(* CoDeSys 2.3.10.0 project: Test.pro *)
(* Libraries: STANDARD.LIB 5.6.98 12:03:02 *)

(* Task configuration *)
TASK Standard (PRIORITY := 0, INTERVAL := T#10ms);
	MAIN();
END_TASK

(* Global variable list: Global_Variables *)
VAR_GLOBAL
	Zielona_1 		AT 	%Q* 	:	 BOOL:= 0;
	Zielona_2 		AT 	%Q* 	:	 BOOL:= 0;
	Zielona_3 		AT 	%Q* 	:	 BOOL:= 0;
	Zielona_4 		AT 	%Q* 	:	 BOOL:= 0;

	Czerwona_1 		AT 	%Q*		:	 BOOL:= 0;
	Czerwona_2 		AT 	%Q*		:	 BOOL:= 0;
	Czerwona_3 		AT	%Q*		:	 BOOL:= 0;
	Czerwona_4 		AT 	%Q*		:	 BOOL:= 0;

	Przycisk_1 		AT 	%I*		:	BOOL;
	Przycisk_2 		AT 	%I*		: 	BOOL;
	Przycisk_3 		AT 	%I*		: 	BOOL;
	Przycisk_4 		AT 	%I*		: 	BOOL;

	RegulatorIn_1 	AT 	%I*		:	INT;
	RegulatorIn_2 	AT 	%I*		:	INT;

	RegulatorOut_1 	AT 	%Q*		:	UDINT;
	RegulatorOut_2 	AT 	%Q*		:	UDINT;

	Scale_1			AT	%Q*		:	INT;
	Scale_2			AT	%Q*		:	INT;

	Enable_1		AT	%Q*		:	BOOL;
	Enable_2		AT 	%Q*		:	BOOL;

(*	Velo_1			AT	%I*		:	LREAL;*)
(*	Velo_2			AT	%I*		:	LREAL;*)
END_VAR

(* Global variable list: TwinCAT_Configuration *)
(* Generated automatically by TwinCAT - (read only) *)
VAR_CONFIG
	.Zielona_1 AT %QX0.0 : BOOL;	(*  ~ {LinkedWith:TIID^Device 2 (EtherCAT (v2.10 only))^Term 1 (EK1100)^Zielone (EL2004)^Channel 1^Output} *)
	.Zielona_2 AT %QX0.1 : BOOL;	(*  ~ {LinkedWith:TIID^Device 2 (EtherCAT (v2.10 only))^Term 1 (EK1100)^Zielone (EL2004)^Channel 2^Output} *)
	.Zielona_3 AT %QX0.2 : BOOL;	(*  ~ {LinkedWith:TIID^Device 2 (EtherCAT (v2.10 only))^Term 1 (EK1100)^Zielone (EL2004)^Channel 3^Output} *)
	.Zielona_4 AT %QX0.3 : BOOL;	(*  ~ {LinkedWith:TIID^Device 2 (EtherCAT (v2.10 only))^Term 1 (EK1100)^Zielone (EL2004)^Channel 4^Output} *)
	.Czerwona_1 AT %QX0.4 : BOOL;	(*  ~ {LinkedWith:TIID^Device 2 (EtherCAT (v2.10 only))^Term 1 (EK1100)^Czerwone (EL2004)^Channel 1^Output} *)
	.Czerwona_2 AT %QX0.5 : BOOL;	(*  ~ {LinkedWith:TIID^Device 2 (EtherCAT (v2.10 only))^Term 1 (EK1100)^Czerwone (EL2004)^Channel 2^Output} *)
	.Czerwona_3 AT %QX0.6 : BOOL;	(*  ~ {LinkedWith:TIID^Device 2 (EtherCAT (v2.10 only))^Term 1 (EK1100)^Czerwone (EL2004)^Channel 3^Output} *)
	.Czerwona_4 AT %QX0.7 : BOOL;	(*  ~ {LinkedWith:TIID^Device 2 (EtherCAT (v2.10 only))^Term 1 (EK1100)^Czerwone (EL2004)^Channel 4^Output} *)
	.Przycisk_1 AT %IX0.0 : BOOL;	(*  ~ {LinkedWith:TIID^Device 2 (EtherCAT (v2.10 only))^Term 1 (EK1100)^Przyciski (EL1004)^Channel 1^Input} *)
	.Przycisk_2 AT %IX0.1 : BOOL;	(*  ~ {LinkedWith:TIID^Device 2 (EtherCAT (v2.10 only))^Term 1 (EK1100)^Przyciski (EL1004)^Channel 2^Input} *)
	.Przycisk_3 AT %IX0.2 : BOOL;	(*  ~ {LinkedWith:TIID^Device 2 (EtherCAT (v2.10 only))^Term 1 (EK1100)^Przyciski (EL1004)^Channel 3^Input} *)
	.Przycisk_4 AT %IX0.3 : BOOL;	(*  ~ {LinkedWith:TIID^Device 2 (EtherCAT (v2.10 only))^Term 1 (EK1100)^Przyciski (EL1004)^Channel 4^Input} *)
	.RegulatorIn_1 AT %IB4 : INT;	(*  ~ {LinkedWith:TIID^Device 2 (EtherCAT (v2.10 only))^Term 1 (EK1100)^Term 6 (EL3102)^Channel 1^Value} *)
	.RegulatorIn_2 AT %IB6 : INT;	(*  ~ {LinkedWith:TIID^Device 2 (EtherCAT (v2.10 only))^Term 1 (EK1100)^Term 6 (EL3102)^Channel 2^Value} *)
	.RegulatorOut_1 AT %QB4 : UDINT;	(*  ~ {LinkedWith:TINC^NC-Task 1 SAF^Axes^Axis 1^Inputs^Axis 1_FromPlc^Override} *)
	.RegulatorOut_2 AT %QB8 : UDINT;	(*  ~ {LinkedWith:TINC^NC-Task 1 SAF^Axes^Axis 2^Inputs^Axis 2_FromPlc^Override} *)
	.Scale_1 AT %QB12 : INT;	(*  ~ {LinkedWith:TIID^Device 2 (EtherCAT (v2.10 only))^Term 1 (EK1100)^Term 2 (EL4132)^Channel 1^Output} *)
	.Scale_2 AT %QB14 : INT;	(*  ~ {LinkedWith:TIID^Device 2 (EtherCAT (v2.10 only))^Term 1 (EK1100)^Term 2 (EL4132)^Channel 2^Output} *)
	.Enable_1 AT %QX16.0 : BOOL;	(*  ~ {LinkedWith:TINC^NC-Task 1 SAF^Axes^Axis 1^Inputs^Axis 1_FromPlc^ControlDWord^Enable;TINC^NC-Task 1 SAF^Axes^Axis 1^Inputs^Axis 1_FromPlc^ControlDWord^FeedEnablePlus;TINC^NC-Task 1 SAF^Axes^Axis 1^Inputs^Axis 1_FromPlc^ControlDWord^FeedEnableMinus} *)
	.Enable_2 AT %QX16.1 : BOOL;	(*  ~ {LinkedWith:TINC^NC-Task 1 SAF^Axes^Axis 2^Inputs^Axis 2_FromPlc^ControlDWord^Enable;TINC^NC-Task 1 SAF^Axes^Axis 2^Inputs^Axis 2_FromPlc^ControlDWord^FeedEnablePlus;TINC^NC-Task 1 SAF^Axes^Axis 2^Inputs^Axis 2_FromPlc^ControlDWord^FeedEnableMinus} *)
END_VAR

(* POU MAIN, ST *)
PROGRAM MAIN
VAR
END_VAR
Czerwona_1 :=  NOT Przycisk_1;
Czerwona_2 :=  NOT Przycisk_2;
Czerwona_3 :=  NOT Przycisk_3;
Czerwona_4 :=  NOT Przycisk_4;

IF Przycisk_1 THEN
	Zielona_1:=  TRUE;
(*	Velo_1 := -600.00;*)
END_IF;

IF Przycisk_2 THEN
	Zielona_2:=  TRUE;
(*	Velo_1 := -100.00;*)
END_IF;

IF Przycisk_3 THEN
	Zielona_3:=  TRUE;
(*	Velo_1 := 100.00;*)
END_IF;

IF Przycisk_4 THEN
	Zielona_4:=  TRUE;
(*	Velo_1 := 600.00;*)
END_IF;

Enable_1 := TRUE;
Enable_2 := TRUE;

Scale_1 := 100;
Scale_2 := 100;

IF (RegulatorIn_1   < 100) AND (RegulatorIn_1   > 0) THEN
	RegulatorOut_1 := RegulatorIn_1 * 10000;
ELSE IF (RegulatorIn_1   > 100) THEN
		RegulatorOut_1 := 100 * 10000;
END_IF;
END_IF;

IF (RegulatorIn_2   < 100) AND (RegulatorIn_2   > 0) THEN
	RegulatorOut_2 := RegulatorIn_2 * 10000;
ELSE IF (RegulatorIn_2   > 100) THEN
		RegulatorOut_2 := 100 * 10000;
END_IF;
END_IF;
END_PROGRAM

(* Visualisation StandState
1 more shapes without text or variables
*)
